// TIA Portal project "PLCtilWinSocket1" (V13)

(* hardware
DEVICE "S7-1200 station_1"  S7-1200 Station
   slot 0: "Rack_0"  Rack  V1.0
   slot 1: "PLC_1"  CPU 1214C DC/DC/DC  6ES7 214-1AG40-0XB0  V4.1
   slot 3: "AQ 1x12BIT_1"  6ES7 232-4HA30-0XB0  V1.0
*)

// ===== PLC "PLC_1"  CPU 1214C DC/DC/DC =====

VAR_GLOBAL   // PLC tag table "Default tag table"
   "EnableForbindelse" AT %I0.0 : Bool;
   "EnableSend" AT %I0.1 : Bool;
   "EnableModtag" AT %I0.2 : Bool;
   "DisableForbindelse" AT %I0.3 : Bool;
END_VAR

DATA_BLOCK "Data"   // DB4
{ S7_Optimized_Access := 'FALSE' }
VERSION : 0.1
   VAR
      ModtagData : Array[0..3] of Char;
      SendData : Array[0..3] of Char;
   END_VAR
BEGIN
END_DATA_BLOCK

DATA_BLOCK "Kommunikationsstyring_DB"   // DB8
{ S7_Optimized_Access := 'FALSE' }
VERSION : 0.1
// stored: InstanceOfName Kommunikationsstyring
"Kommunikationsstyring"
BEGIN
END_DATA_BLOCK

// folder: System blocks/Program resources

DATA_BLOCK "PLC_1_Connection_DB"   // DB2
{ S7_Optimized_Access := 'FALSE' }
AUTHOR : SIMATIC
FAMILY : MC7Plus
NAME : TC_IP_v4
VERSION : 1.0
// stored: InstanceOfName ?
"?"
BEGIN
END_DATA_BLOCK

DATA_BLOCK "IEC_Timer_0_DB"   // DB7
{ S7_Optimized_Access := 'FALSE' }
AUTHOR : Simatic
FAMILY : IEC
NAME : IEC_TMR
VERSION : 1.0
// stored: InstanceOfName ?
"?"
BEGIN
END_DATA_BLOCK

// folder: (top level)

FUNCTION_BLOCK "Kommunikationsstyring"   // FB1, LAD
{ S7_Optimized_Access := 'FALSE' }
VERSION : 0.1
   VAR_TEMP   // added for the SCL form of the ladder/FBD networks
      _w1 : Bool;
   END_VAR
BEGIN

REGION Network 1: Step 0 - Enable forbindelse
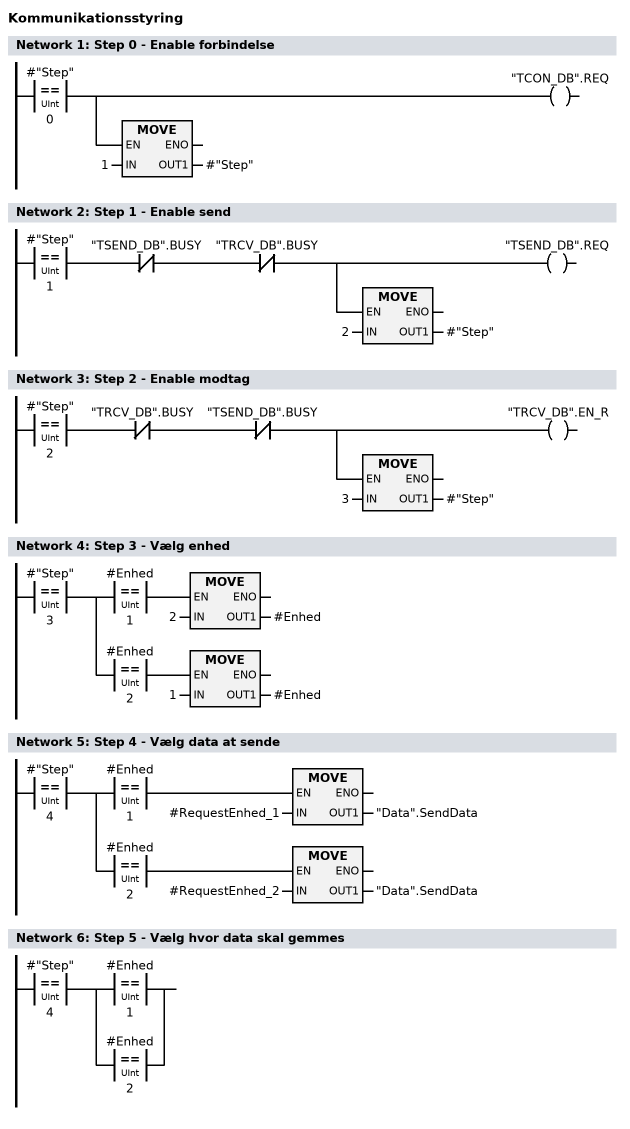
   RUNG wire#powerrail
      { S7_Templates := "SrcType := UInt" } EQ_Contact(in1 := #"Step", in2 := 0)
      wire#w1
      Coil( "TCON_DB".REQ )
   END_RUNG
   RUNG wire#w1
      Move(in := 1, out1 => #"Step")
   END_RUNG
   // the same network as SCL:
   "TCON_DB".REQ := #"Step" = 0;
   IF "TCON_DB".REQ THEN #"Step" := 1; END_IF;
END_REGION

REGION Network 2: Step 1 - Enable send
   RUNG wire#powerrail
      { S7_Templates := "SrcType := UInt" } EQ_Contact(in1 := #"Step", in2 := 1)
      I_Contact( "TSEND_DB".BUSY )
      I_Contact( "TRCV_DB".BUSY )
      wire#w1
      Coil( "TSEND_DB".REQ )
   END_RUNG
   RUNG wire#w1
      Move(in := 2, out1 => #"Step")
   END_RUNG
   // the same network as SCL:
   "TSEND_DB".REQ := (#"Step" = 1) AND NOT "TSEND_DB".BUSY AND NOT "TRCV_DB".BUSY;
   IF "TSEND_DB".REQ THEN #"Step" := 2; END_IF;
END_REGION

REGION Network 3: Step 2 - Enable modtag
   RUNG wire#powerrail
      { S7_Templates := "SrcType := UInt" } EQ_Contact(in1 := #"Step", in2 := 2)
      I_Contact( "TRCV_DB".BUSY )
      I_Contact( "TSEND_DB".BUSY )
      wire#w1
      Coil( "TRCV_DB".EN_R )
   END_RUNG
   RUNG wire#w1
      Move(in := 3, out1 => #"Step")
   END_RUNG
   // the same network as SCL:
   "TRCV_DB".EN_R := (#"Step" = 2) AND NOT "TRCV_DB".BUSY AND NOT "TSEND_DB".BUSY;
   IF "TRCV_DB".EN_R THEN #"Step" := 3; END_IF;
END_REGION

REGION Network 4: Step 3 - Vælg enhed
   RUNG wire#powerrail
      { S7_Templates := "SrcType := UInt" } EQ_Contact(in1 := #"Step", in2 := 3)
      wire#w1
      { S7_Templates := "SrcType := UInt" } EQ_Contact(in1 := #Enhed, in2 := 1)
      Move(in := 2, out1 => #Enhed)
   END_RUNG
   RUNG wire#w1
      { S7_Templates := "SrcType := UInt" } EQ_Contact(in1 := #Enhed, in2 := 2)
      Move(in := 1, out1 => #Enhed)
   END_RUNG
   // the same network as SCL:
   #_w1 := #"Step" = 3;
   IF #_w1 AND (#Enhed = 1) THEN #Enhed := 2; END_IF;
   IF #_w1 AND (#Enhed = 2) THEN #Enhed := 1; END_IF;
END_REGION

REGION Network 5: Step 4 - Vælg data at sende
   RUNG wire#powerrail
      { S7_Templates := "SrcType := UInt" } EQ_Contact(in1 := #"Step", in2 := 4)
      wire#w1
      { S7_Templates := "SrcType := UInt" } EQ_Contact(in1 := #Enhed, in2 := 1)
      Move(in := #RequestEnhed_1, out1 => "Data".SendData)
   END_RUNG
   RUNG wire#w1
      { S7_Templates := "SrcType := UInt" } EQ_Contact(in1 := #Enhed, in2 := 2)
      Move(in := #RequestEnhed_2, out1 => "Data".SendData)
   END_RUNG
   // the same network as SCL:
   #_w1 := #"Step" = 4;
   IF #_w1 AND (#Enhed = 1) THEN "Data".SendData := #RequestEnhed_1; END_IF;
   IF #_w1 AND (#Enhed = 2) THEN "Data".SendData := #RequestEnhed_2; END_IF;
END_REGION

REGION Network 6: Step 5 - Vælg hvor data skal gemmes
END_REGION
END_FUNCTION_BLOCK

FUNCTION "OpretForbindelse" : Void   // FC1, LAD
{ S7_Optimized_Access := 'FALSE' }
VERSION : 0.1
BEGIN

REGION Network 1
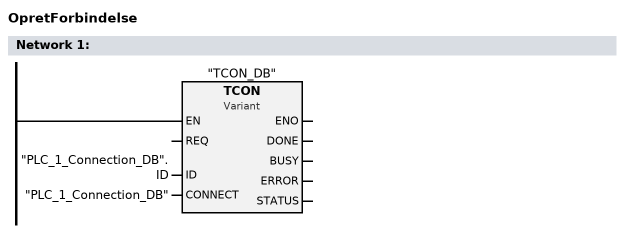
   "TCON_DB"(ID := "PLC_1_Connection_DB".ID, CONNECT := "PLC_1_Connection_DB");   // TCON
END_REGION
END_FUNCTION

FUNCTION "Modtag" : Void   // FC2, LAD
{ S7_Optimized_Access := 'FALSE' }
VERSION : 0.1
BEGIN

REGION Network 1: Modtag data
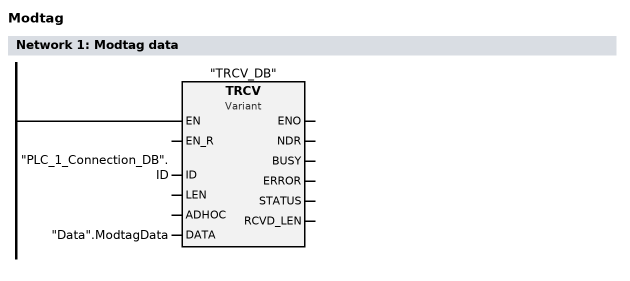
   "TRCV_DB"(ID := "PLC_1_Connection_DB".ID, DATA := "Data".ModtagData);   // TRCV
END_REGION
END_FUNCTION

FUNCTION "Send" : Void   // FC3, LAD
{ S7_Optimized_Access := 'FALSE' }
VERSION : 0.1
BEGIN

REGION Network 1
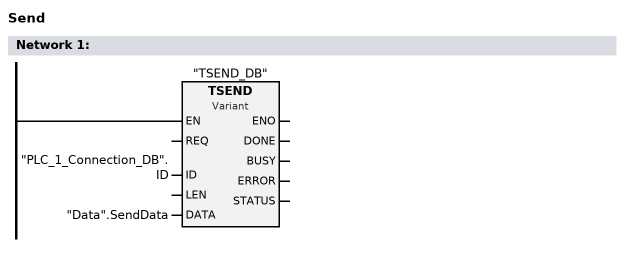
   "TSEND_DB"(ID := "PLC_1_Connection_DB".ID, DATA := "Data".SendData);   // TSEND
END_REGION
END_FUNCTION

FUNCTION "AfslutForbindelse" : Void   // FC4, LAD
{ S7_Optimized_Access := 'FALSE' }
VERSION : 0.1
BEGIN

REGION Network 1
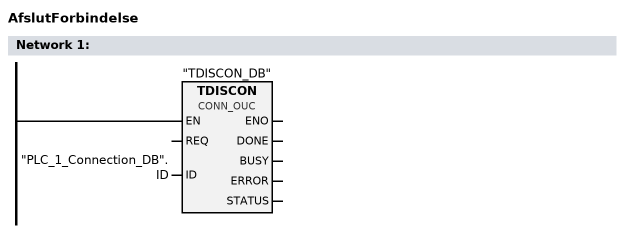
   "TDISCON_DB"(ID := "PLC_1_Connection_DB".ID);   // TDISCON
END_REGION
END_FUNCTION

ORGANIZATION_BLOCK "Main"   // OB1, LAD, ProgramCycle
TITLE = "Main Program Sweep (Cycle)"
{ S7_Optimized_Access := 'FALSE' }
VERSION : 0.1
BEGIN

REGION Network 1: Opret forbindelse
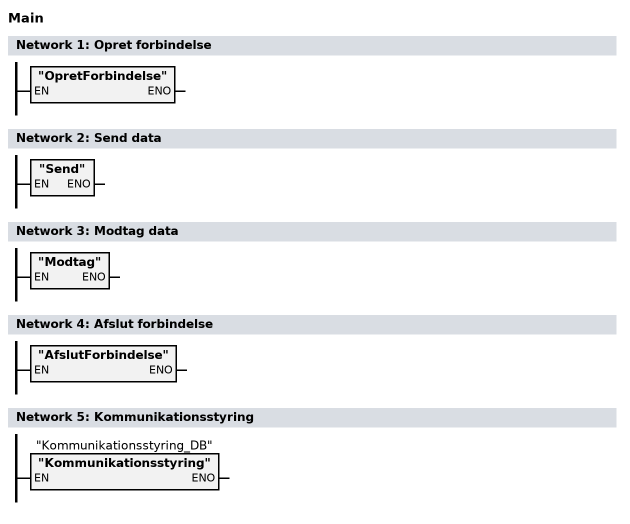
   RUNG wire#powerrail
      "OpretForbindelse"()
   END_RUNG
   // the same network as SCL:
   "OpretForbindelse"();
END_REGION

REGION Network 2: Send data
   RUNG wire#powerrail
      "Send"()
   END_RUNG
   // the same network as SCL:
   "Send"();
END_REGION

REGION Network 3: Modtag data
   RUNG wire#powerrail
      "Modtag"()
   END_RUNG
   // the same network as SCL:
   "Modtag"();
END_REGION

REGION Network 4: Afslut forbindelse
   RUNG wire#powerrail
      "AfslutForbindelse"()
   END_RUNG
   // the same network as SCL:
   "AfslutForbindelse"();
END_REGION

REGION Network 5: Kommunikationsstyring
   RUNG wire#powerrail
      "Kommunikationsstyring_DB"()
   END_RUNG
   // the same network as SCL:
   "Kommunikationsstyring_DB"();   // "Kommunikationsstyring"
END_REGION
END_ORGANIZATION_BLOCK